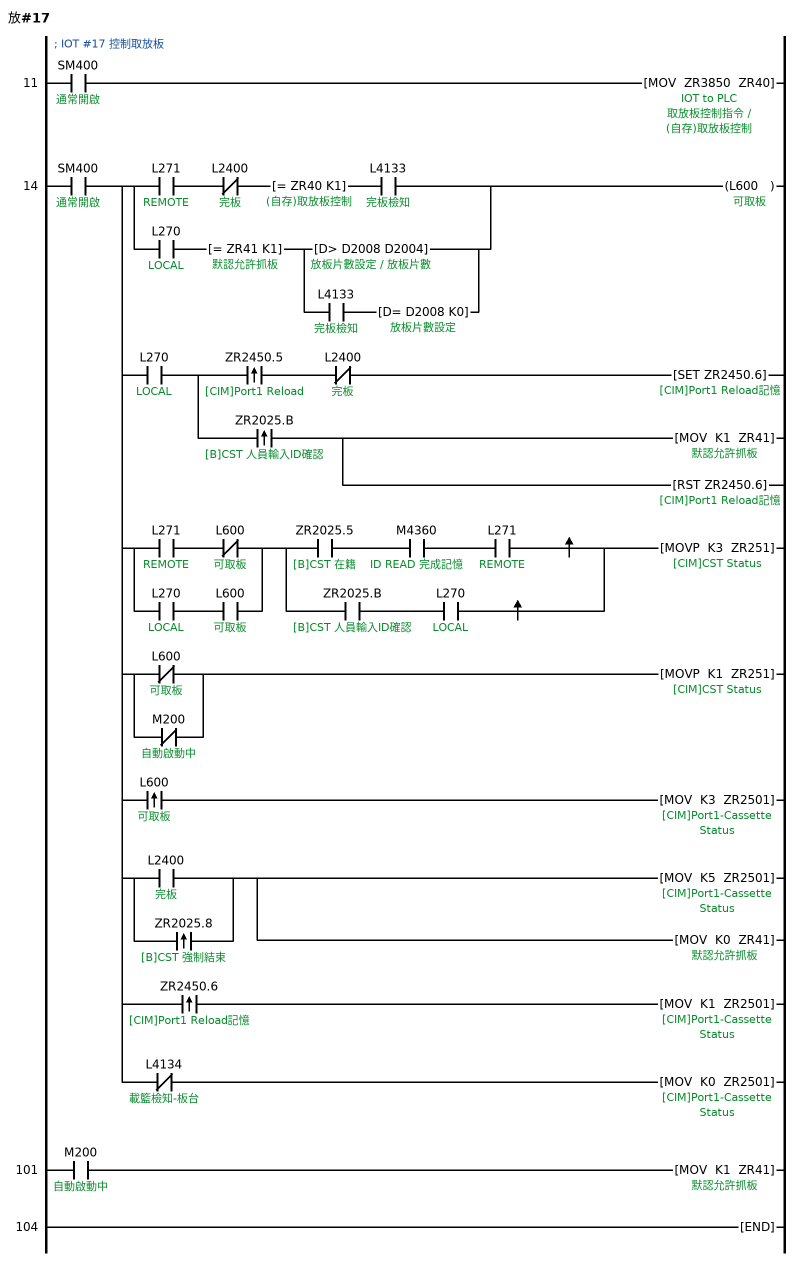
; IOT #17 控制取放板
11    LD      SM400  ; 通常開啟
      MOV     ZR3850 ZR40  ; IOT to PLC 取放板控制指令 / (自存)取放板控制
14    LD      SM400  ; 通常開啟
      MPS
      LD      L271  ; REMOTE
      ANI     L2400  ; 完板
      AND=    ZR40 K1  ; (自存)取放板控制
      AND     L4133  ; 完板檢知
      LD      L270  ; LOCAL
      AND=    ZR41 K1  ; 默認允許抓板
      LDD>    D2008 D2004  ; 放板片數設定 / 放板片數
      LD      L4133  ; 完板檢知
      ANDD=   D2008 K0  ; 放板片數設定
      ORB
      ANB
      ORB
      ANB
      OUT     L600  ; 可取板
      MRD
      AND     L270  ; LOCAL
      MPS
      ANDP    ZR2450.5  ; [CIM]Port1 Reload
      ANI     L2400  ; 完板
      SET     ZR2450.6  ; [CIM]Port1 Reload記憶
      MPP
      ANDP    ZR2025.B  ; [B]CST 人員輸入ID確認
      MOV     K1 ZR41
      RST     ZR2450.6  ; [CIM]Port1 Reload記憶
      MRD
      LD      L271  ; REMOTE
      ANI     L600  ; 可取板
      LD      L270  ; LOCAL
      AND     L600  ; 可取板
      ORB
      ANB
      LD      ZR2025.5  ; [B]CST 在籍
      AND     M4360  ; ID READ 完成記憶
      AND     L271  ; REMOTE
      MEP
      LD      ZR2025.B  ; [B]CST 人員輸入ID確認
      AND     L270  ; LOCAL
      MEP
      ORB
      ANB
      MOVP    K3 ZR251  ; [CIM]CST Status
      MRD
      LDI     L600  ; 可取板
      ORI     M200  ; 自動啟動中
      ANB
      MOVP    K1 ZR251
      MRD
      ANDP    L600  ; 可取板
      MOV     K3 ZR2501  ; [CIM]Port1-Cassette Status
      MRD
      LD      L2400  ; 完板
      ORP     ZR2025.8  ; [B]CST 強制結束
      ANB
      MOV     K5 ZR2501
      MOV     K0 ZR41
      MRD
      ANDP    ZR2450.6  ; [CIM]Port1 Reload記憶
      MOV     K1 ZR2501
      MPP
      ANI     L4134  ; 載籃檢知-板台
      MOV     K0 ZR2501
101   LD      M200  ; 自動啟動中
      MOV     K1 ZR41
104   END
END_PROGRAM

PROGRAM M98
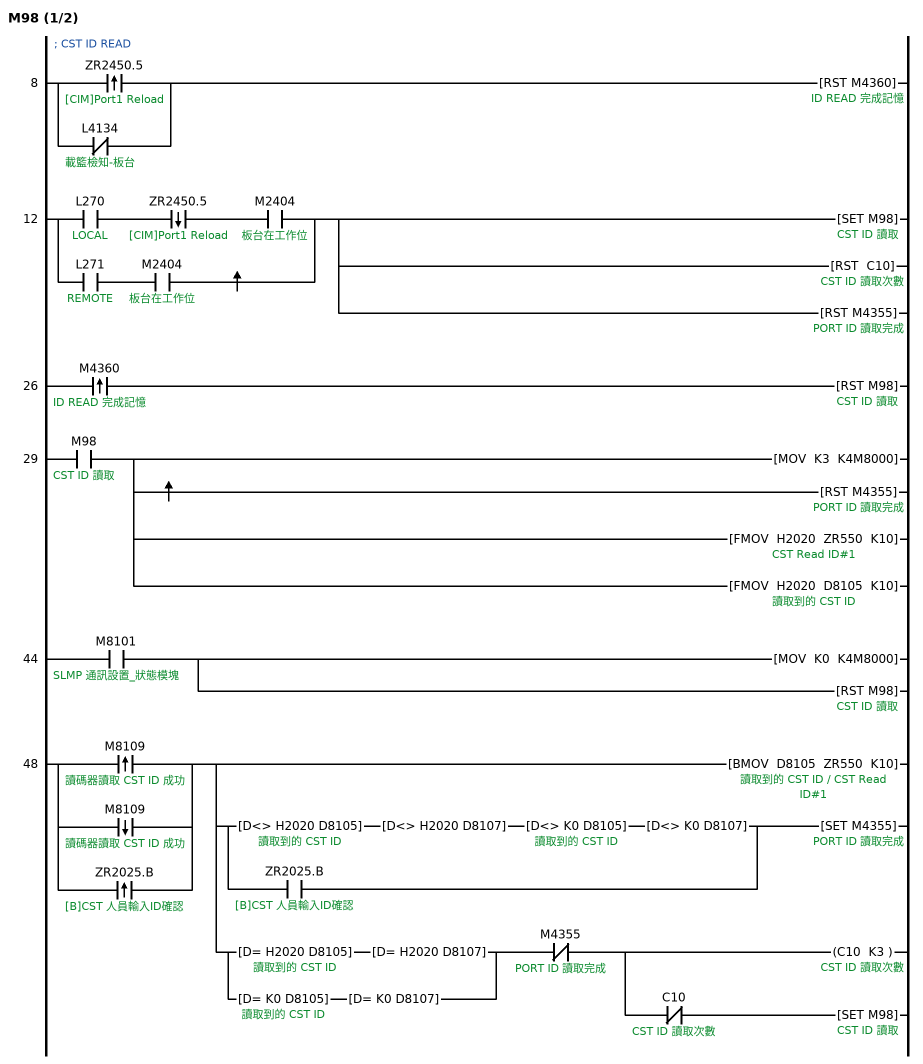
; CST ID READ
8     LDP     ZR2450.5  ; [CIM]Port1 Reload
      ORI     L4134  ; 載籃檢知-板台
      RST     M4360  ; ID READ 完成記憶
12    LD      L270  ; LOCAL
      ANDF    ZR2450.5  ; [CIM]Port1 Reload
      AND     M2404  ; 板台在工作位
      LD      L271  ; REMOTE
      AND     M2404  ; 板台在工作位
      MEP
      ORB
      SET     M98  ; CST ID 讀取
      RST     C10  ; CST ID 讀取次數
      RST     M4355  ; PORT ID 讀取完成
26    LDP     M4360  ; ID READ 完成記憶
      RST     M98  ; CST ID 讀取
29    LD      M98  ; CST ID 讀取
      MOV     K3 K4M8000  ; SLMP 通訊設置_控制模塊
      MPS
      MEP
      RST     M4355  ; PORT ID 讀取完成
      MPP
      FMOV    H2020 ZR550 K10  ; CST Read ID#1
      FMOV    H2020 D8105 K10  ; 讀取到的 CST ID
44    LD      M8101  ; SLMP 通訊設置_狀態模塊
      MOV     K0 K4M8000
      RST     M98  ; CST ID 讀取
48    LDP     M8109  ; 讀碼器讀取 CST ID 成功
      ORF     M8109  ; 讀碼器讀取 CST ID 成功
      ORP     ZR2025.B  ; [B]CST 人員輸入ID確認
      BMOV    D8105 ZR550 K10
      MPS
      LDD<>   H2020 D8105  ; 讀取到的 CST ID
      ANDD<>  H2020 D8107
      ANDD<>  K0 D8105  ; 讀取到的 CST ID
      ANDD<>  K0 D8107
      OR      ZR2025.B  ; [B]CST 人員輸入ID確認
      ANB
      SET     M4355  ; PORT ID 讀取完成
      MPP
      LDD=    H2020 D8105  ; 讀取到的 CST ID
      ANDD=   H2020 D8107
      LDD=    K0 D8105  ; 讀取到的 CST ID
      ANDD=   K0 D8107
      ORB
      ANB
      ANI     M4355  ; PORT ID 讀取完成
      OUT     C10 K3  ; CST ID 讀取次數
      ANI     C10  ; CST ID 讀取次數
      SET     M98  ; CST ID 讀取
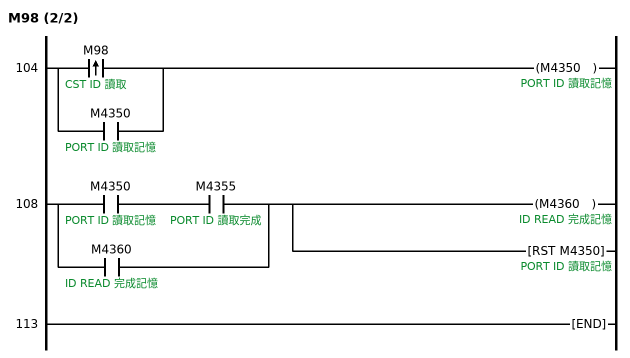
104   LDP     M98  ; CST ID 讀取
      OR      M4350  ; PORT ID 讀取記憶
      OUT     M4350  ; PORT ID 讀取記憶
108   LD      M4350  ; PORT ID 讀取記憶
      AND     M4355  ; PORT ID 讀取完成
      OR      M4360  ; ID READ 完成記憶
      OUT     M4360  ; ID READ 完成記憶
      RST     M4350  ; PORT ID 讀取記憶
113   END
END_PROGRAM

PROGRAM 低M90
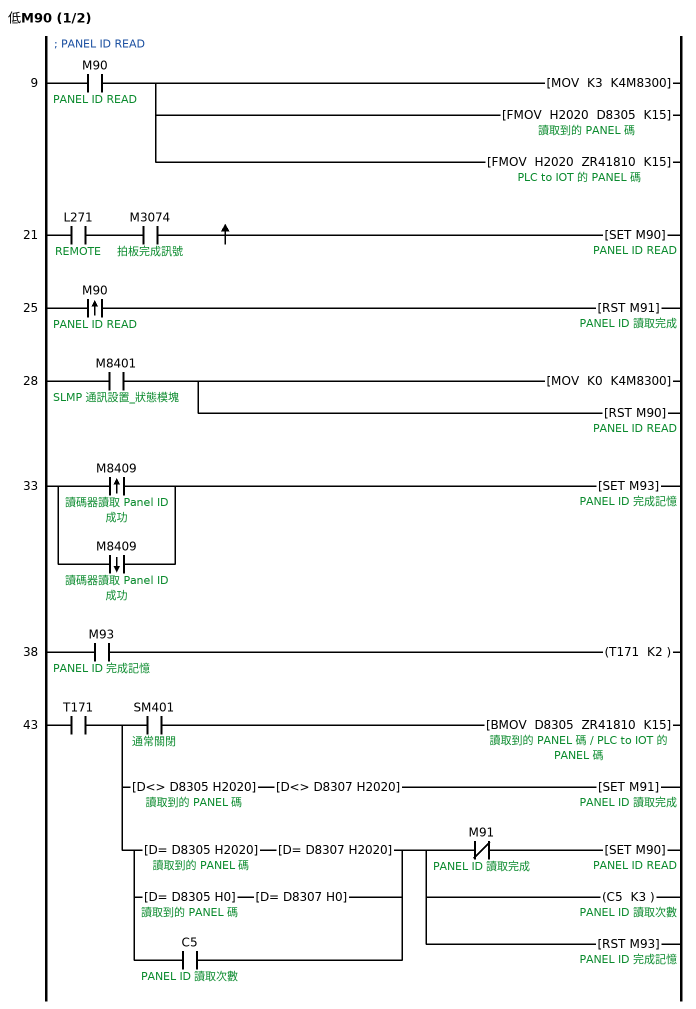
; PANEL ID READ
9     LD      M90  ; PANEL ID READ
      MOV     K3 K4M8300  ; SLMP 通訊設置_控制模塊
      FMOV    H2020 D8305 K15  ; 讀取到的 PANEL 碼
      FMOV    H2020 ZR41810 K15  ; PLC to IOT 的 PANEL 碼
21    LD      L271  ; REMOTE
      AND     M3074  ; 拍板完成訊號
      MEP
      SET     M90  ; PANEL ID READ
25    LDP     M90  ; PANEL ID READ
      RST     M91  ; PANEL ID 讀取完成
28    LD      M8401  ; SLMP 通訊設置_狀態模塊
      MOV     K0 K4M8300
      RST     M90  ; PANEL ID READ
33    LDP     M8409  ; 讀碼器讀取 Panel ID 成功
      ORF     M8409  ; 讀碼器讀取 Panel ID 成功
      SET     M93  ; PANEL ID 完成記憶
38    LD      M93  ; PANEL ID 完成記憶
      OUT     T171 K2
43    LD      T171
      MPS
      AND     SM401  ; 通常關閉
      BMOV    D8305 ZR41810 K15
      MRD
      ANDD<>  D8305 H2020  ; 讀取到的 PANEL 碼
      ANDD<>  D8307 H2020
      SET     M91  ; PANEL ID 讀取完成
      MPP
      LDD=    D8305 H2020  ; 讀取到的 PANEL 碼
      ANDD=   D8307 H2020
      LDD=    D8305 H0  ; 讀取到的 PANEL 碼
      ANDD=   D8307 H0
      ORB
      OR      C5  ; PANEL ID 讀取次數
      ANB
      MPS
      ANI     M91  ; PANEL ID 讀取完成
      SET     M90  ; PANEL ID READ
      MPP
      OUT     C5 K3  ; PANEL ID 讀取次數
      RST     M93  ; PANEL ID 完成記憶
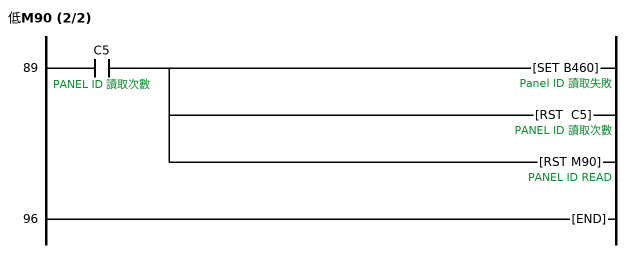
89    LD      C5  ; PANEL ID 讀取次數
      SET     B460  ; Panel ID 讀取失敗
      RST     C5  ; PANEL ID 讀取次數
      RST     M90  ; PANEL ID READ
96    END
END_PROGRAM

PROGRAM 高M90
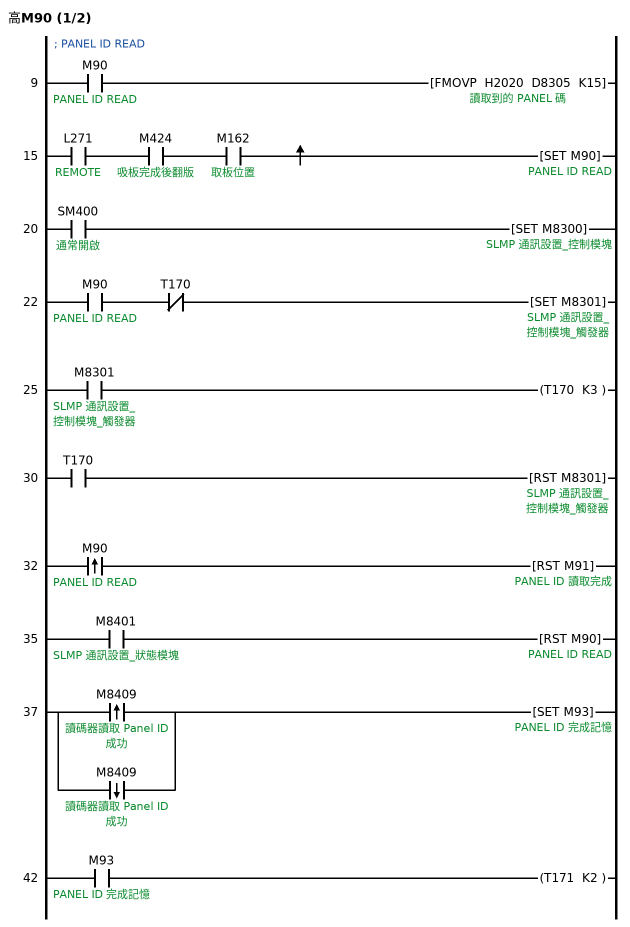
; PANEL ID READ
9     LD      M90  ; PANEL ID READ
      FMOVP   H2020 D8305 K15  ; 讀取到的 PANEL 碼
15    LD      L271  ; REMOTE
      AND     M424  ; 吸板完成後翻版
      AND     M162  ; 取板位置
      MEP
      SET     M90  ; PANEL ID READ
20    LD      SM400  ; 通常開啟
      SET     M8300  ; SLMP 通訊設置_控制模塊
22    LD      M90  ; PANEL ID READ
      ANI     T170
      SET     M8301  ; SLMP 通訊設置_控制模塊_觸發器
25    LD      M8301  ; SLMP 通訊設置_控制模塊_觸發器
      OUT     T170 K3
30    LD      T170
      RST     M8301  ; SLMP 通訊設置_控制模塊_觸發器
32    LDP     M90  ; PANEL ID READ
      RST     M91  ; PANEL ID 讀取完成
35    LD      M8401  ; SLMP 通訊設置_狀態模塊
      RST     M90  ; PANEL ID READ
37    LDP     M8409  ; 讀碼器讀取 Panel ID 成功
      ORF     M8409  ; 讀碼器讀取 Panel ID 成功
      SET     M93  ; PANEL ID 完成記憶
42    LD      M93  ; PANEL ID 完成記憶
      OUT     T171 K2
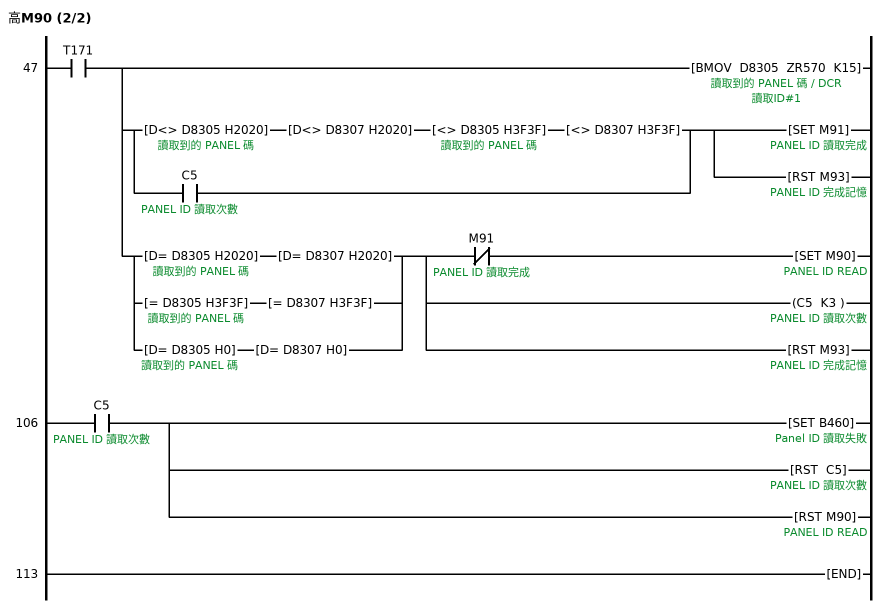
47    LD      T171
      BMOV    D8305 ZR570 K15  ; DCR 讀取ID#1
      MPS
      LDD<>   D8305 H2020  ; 讀取到的 PANEL 碼
      ANDD<>  D8307 H2020
      AND<>   D8305 H3F3F  ; 讀取到的 PANEL 碼
      AND<>   D8307 H3F3F
      OR      C5  ; PANEL ID 讀取次數
      ANB
      SET     M91  ; PANEL ID 讀取完成
      RST     M93  ; PANEL ID 完成記憶
      MPP
      LDD=    D8305 H2020  ; 讀取到的 PANEL 碼
      ANDD=   D8307 H2020
      LD=     D8305 H3F3F  ; 讀取到的 PANEL 碼
      AND=    D8307 H3F3F
      ORB
      LDD=    D8305 H0  ; 讀取到的 PANEL 碼
      ANDD=   D8307 H0
      ORB
      ANB
      MPS
      ANI     M91  ; PANEL ID 讀取完成
      SET     M90  ; PANEL ID READ
      MPP
      OUT     C5 K3  ; PANEL ID 讀取次數
      RST     M93  ; PANEL ID 完成記憶
106   LD      C5  ; PANEL ID 讀取次數
      SET     B460  ; Panel ID 讀取失敗
      RST     C5  ; PANEL ID 讀取次數
      RST     M90  ; PANEL ID READ
113   END
END_PROGRAM

PROGRAM M350
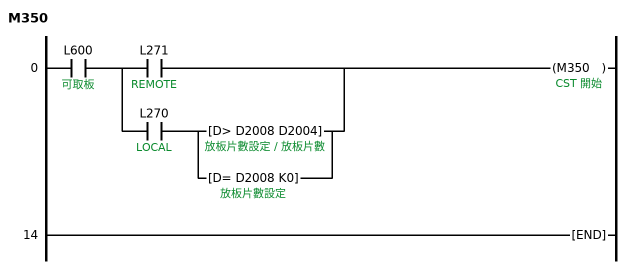
0     LD      L600  ; 可取板
      LD      L271  ; REMOTE
      LD      L270  ; LOCAL
      LDD>    D2008 D2004  ; 放板片數設定 / 放板片數
      ORD=    D2008 K0  ; 放板片數設定
      ANB
      ORB
      ANB
      OUT     M350  ; CST 開始
14    END
END_PROGRAM

PROGRAM M350例
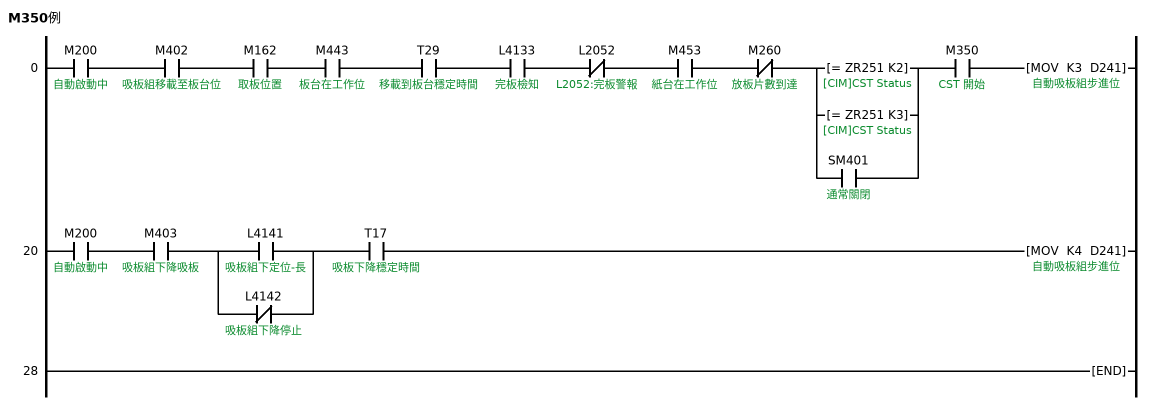
0     LD      M200  ; 自動啟動中
      AND     M402  ; 吸板組移載至板台位
      AND     M162  ; 取板位置
      AND     M443  ; 板台在工作位
      AND     T29  ; 移載到板台穩定時間
      AND     L4133  ; 完板檢知
      ANI     L2052  ; L2052:完板警報
      AND     M453  ; 紙台在工作位
      ANI     M260  ; 放板片數到達
      LD=     ZR251 K2  ; [CIM]CST Status
      OR=     ZR251 K3  ; [CIM]CST Status
      OR      SM401  ; 通常關閉
      ANB
      AND     M350  ; CST 開始
      MOV     K3 D241  ; 自動吸板組步進位
20    LD      M200  ; 自動啟動中
      AND     M403  ; 吸板組下降吸板
      LD      L4141  ; 吸板組下定位-長
      ORI     L4142  ; 吸板組下降停止
      ANB
      AND     T17  ; 吸板下降穩定時間
      MOV     K4 D241
28    END
END_PROGRAM

PROGRAM 中#14
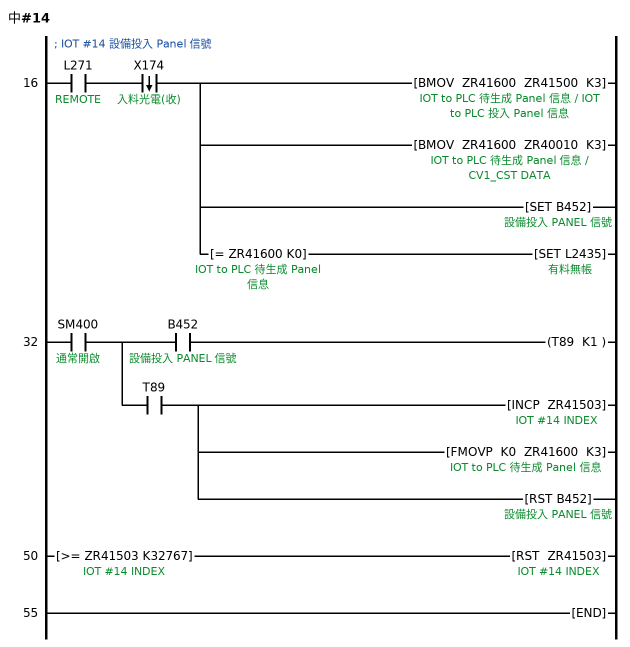
; IOT #14 設備投入 Panel 信號
16    LD      L271  ; REMOTE
      ANDF    X174  ; 入料光電(收)
      BMOV    ZR41600 ZR41500 K3  ; IOT to PLC 待生成 Panel 信息 / IOT to PLC 投入 Panel 信息
      BMOV    ZR41600 ZR40010 K3  ; CV1_CST DATA
      SET     B452  ; 設備投入 PANEL 信號
      AND=    ZR41600 K0  ; IOT to PLC 待生成 Panel 信息
      SET     L2435  ; 有料無帳
32    LD      SM400  ; 通常開啟
      MPS
      AND     B452  ; 設備投入 PANEL 信號
      OUT     T89 K1
      MPP
      AND     T89
      INCP    ZR41503  ; IOT #14 INDEX
      FMOVP   K0 ZR41600 K3
      RST     B452  ; 設備投入 PANEL 信號
50    LD>=    ZR41503 K32767  ; IOT #14 INDEX
      RST     ZR41503  ; IOT #14 INDEX
55    END
END_PROGRAM

PROGRAM 中#15
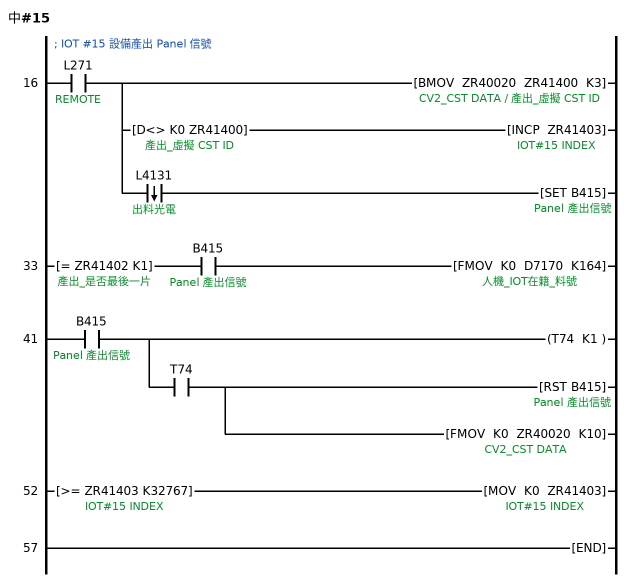
; IOT #15 設備產出 Panel 信號
16    LD      L271  ; REMOTE
      BMOV    ZR40020 ZR41400 K3  ; CV2_CST DATA / 產出_虛擬 CST ID
      MPS
      ANDD<>  K0 ZR41400  ; 產出_虛擬 CST ID
      INCP    ZR41403  ; IOT#15 INDEX
      MPP
      ANDF    L4131  ; 出料光電
      SET     B415  ; Panel 產出信號
33    LD=     ZR41402 K1  ; 產出_是否最後一片
      AND     B415  ; Panel 產出信號
      FMOV    K0 D7170 K164  ; 人機_IOT在籍_料號
41    LD      B415  ; Panel 產出信號
      OUT     T74 K1
      AND     T74
      RST     B415  ; Panel 產出信號
      FMOV    K0 ZR40020 K10
52    LD>=    ZR41403 K32767  ; IOT#15 INDEX
      MOV     K0 ZR41403
57    END
END_PROGRAM

PROGRAM 中#12#13
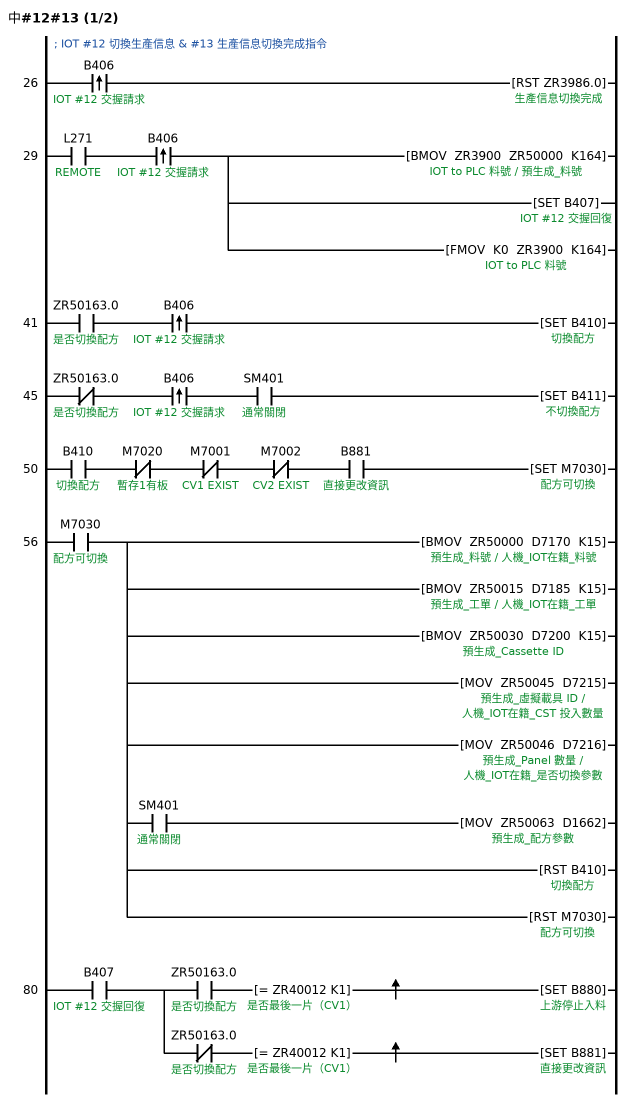
; IOT #12 切換生產信息 & #13 生產信息切換完成指令
26    LDP     B406  ; IOT #12 交握請求
      RST     ZR3986.0  ; 生產信息切換完成
29    LD      L271  ; REMOTE
      ANDP    B406  ; IOT #12 交握請求
      BMOV    ZR3900 ZR50000 K164  ; IOT to PLC 料號 / 預生成_料號
      SET     B407  ; IOT #12 交握回復
      FMOV    K0 ZR3900 K164
41    LD      ZR50163.0  ; 是否切換配方
      ANDP    B406  ; IOT #12 交握請求
      SET     B410  ; 切換配方
45    LDI     ZR50163.0  ; 是否切換配方
      ANDP    B406  ; IOT #12 交握請求
      AND     SM401  ; 通常關閉
      SET     B411  ; 不切換配方
50    LD      B410  ; 切換配方
      ANI     M7020  ; 暫存1有板
      ANI     M7001  ; CV1 EXIST
      ANI     M7002  ; CV2 EXIST
      AND     B881  ; 直接更改資訊
      SET     M7030  ; 配方可切換
56    LD      M7030  ; 配方可切換
      BMOV    ZR50000 D7170 K15  ; 人機_IOT在籍_料號
      BMOV    ZR50015 D7185 K15  ; 預生成_工單 / 人機_IOT在籍_工單
      BMOV    ZR50030 D7200 K15  ; 預生成_Cassette ID
      MOV     ZR50045 D7215  ; 預生成_虛擬載具 ID / 人機_IOT在籍_CST 投入數量
      MOV     ZR50046 D7216  ; 預生成_Panel 數量 / 人機_IOT在籍_是否切換參數
      MPS
      AND     SM401  ; 通常關閉
      MOV     ZR50063 D1662  ; 預生成_配方參數
      MPP
      RST     B410  ; 切換配方
      RST     M7030  ; 配方可切換
80    LD      B407  ; IOT #12 交握回復
      MPS
      AND     ZR50163.0  ; 是否切換配方
      AND=    ZR40012 K1  ; 是否最後一片（CV1）
      MEP
      SET     B880  ; 上游停止入料
      MPP
      ANI     ZR50163.0  ; 是否切換配方
      AND=    ZR40012 K1  ; 是否最後一片（CV1）
      MEP
      SET     B881  ; 直接更改資訊
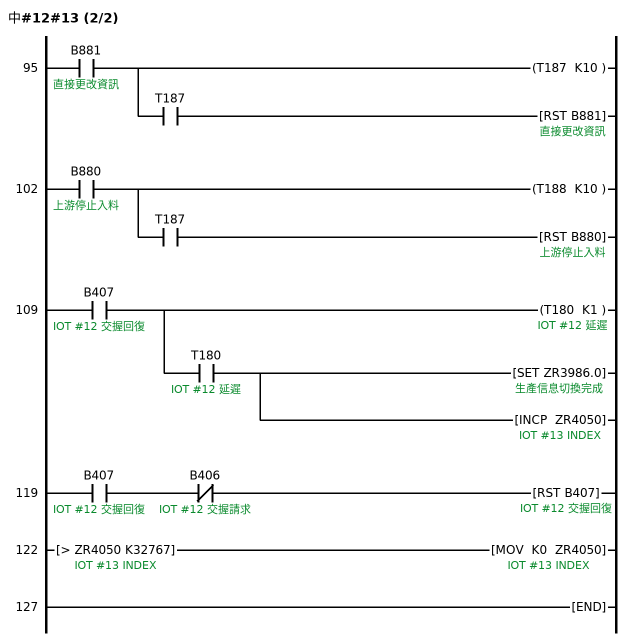
95    LD      B881  ; 直接更改資訊
      OUT     T187 K10
      AND     T187
      RST     B881  ; 直接更改資訊
102   LD      B880  ; 上游停止入料
      OUT     T188 K10
      AND     T187
      RST     B880  ; 上游停止入料
109   LD      B407  ; IOT #12 交握回復
      OUT     T180 K1  ; IOT #12 延遲
      AND     T180  ; IOT #12 延遲
      SET     ZR3986.0  ; 生產信息切換完成
      INCP    ZR4050  ; IOT #13 INDEX
119   LD      B407  ; IOT #12 交握回復
      ANI     B406  ; IOT #12 交握請求
      RST     B407  ; IOT #12 交握回復
122   LD>     ZR4050 K32767  ; IOT #13 INDEX
      MOV     K0 ZR4050
127   END
END_PROGRAM

PROGRAM 附
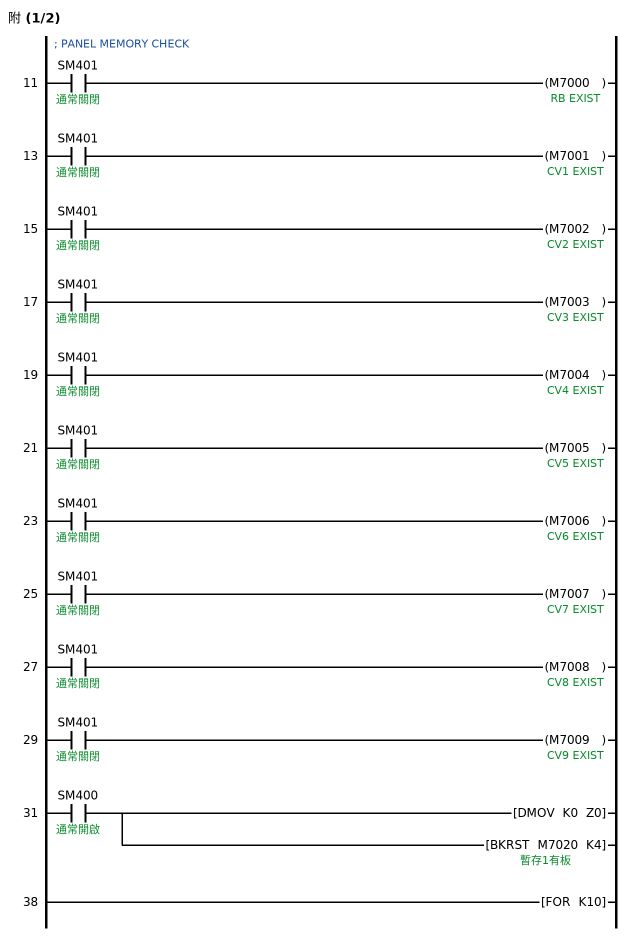
; PANEL MEMORY CHECK
11    LD      SM401  ; 通常關閉
      OUT     M7000  ; RB EXIST
13    LD      SM401  ; 通常關閉
      OUT     M7001  ; CV1 EXIST
15    LD      SM401  ; 通常關閉
      OUT     M7002  ; CV2 EXIST
17    LD      SM401  ; 通常關閉
      OUT     M7003  ; CV3 EXIST
19    LD      SM401  ; 通常關閉
      OUT     M7004  ; CV4 EXIST
21    LD      SM401  ; 通常關閉
      OUT     M7005  ; CV5 EXIST
23    LD      SM401  ; 通常關閉
      OUT     M7006  ; CV6 EXIST
25    LD      SM401  ; 通常關閉
      OUT     M7007  ; CV7 EXIST
27    LD      SM401  ; 通常關閉
      OUT     M7008  ; CV8 EXIST
29    LD      SM401  ; 通常關閉
      OUT     M7009  ; CV9 EXIST
31    LD      SM400  ; 通常開啟
      DMOV    K0 Z0
      BKRST   M7020 K4  ; 暫存1有板
38    FOR     K10
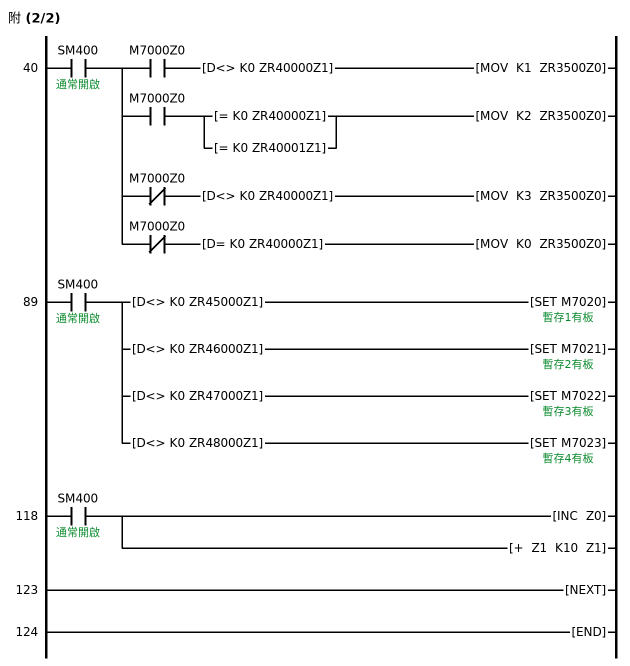
40    LD      SM400  ; 通常開啟
      MPS
      AND     M7000Z0
      ANDD<>  K0 ZR40000Z1
      MOV     K1 ZR3500Z0
      MRD
      AND     M7000Z0
      LD=     K0 ZR40000Z1
      OR=     K0 ZR40001Z1
      ANB
      MOV     K2 ZR3500Z0
      MRD
      ANI     M7000Z0
      ANDD<>  K0 ZR40000Z1
      MOV     K3 ZR3500Z0
      MPP
      ANI     M7000Z0
      ANDD=   K0 ZR40000Z1
      MOV     K0 ZR3500Z0
89    LD      SM400  ; 通常開啟
      MPS
      ANDD<>  K0 ZR45000Z1
      SET     M7020  ; 暫存1有板
      MRD
      ANDD<>  K0 ZR46000Z1
      SET     M7021  ; 暫存2有板
      MRD
      ANDD<>  K0 ZR47000Z1
      SET     M7022  ; 暫存3有板
      MPP
      ANDD<>  K0 ZR48000Z1
      SET     M7023  ; 暫存4有板
118   LD      SM400  ; 通常開啟
      INC     Z0
      +       Z1 K10 Z1
123   NEXT
124   END
END_PROGRAM

PROGRAM FIFO
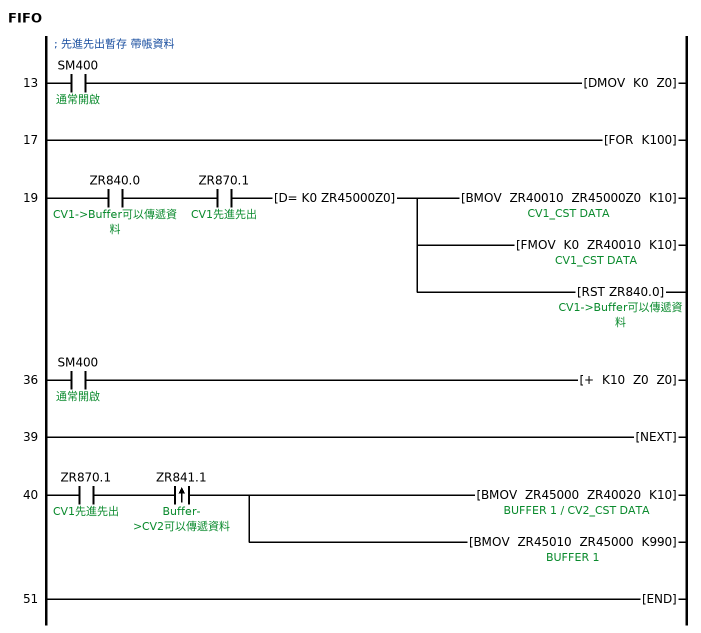
; 先進先出暫存 帶帳資料
13    LD      SM400  ; 通常開啟
      DMOV    K0 Z0
17    FOR     K100
19    LD      ZR840.0  ; CV1->Buffer可以傳遞資料
      AND     ZR870.1  ; CV1先進先出
      ANDD=   K0 ZR45000Z0
      BMOV    ZR40010 ZR45000Z0 K10  ; CV1_CST DATA
      FMOV    K0 ZR40010 K10
      RST     ZR840.0  ; CV1->Buffer可以傳遞資料
36    LD      SM400  ; 通常開啟
      +       K10 Z0 Z0
39    NEXT
40    LD      ZR870.1  ; CV1先進先出
      ANDP    ZR841.1  ; Buffer->CV2可以傳遞資料
      BMOV    ZR45000 ZR40020 K10  ; BUFFER 1 / CV2_CST DATA
      BMOV    ZR45010 ZR45000 K990
51    END
END_PROGRAM

PROGRAM FILO
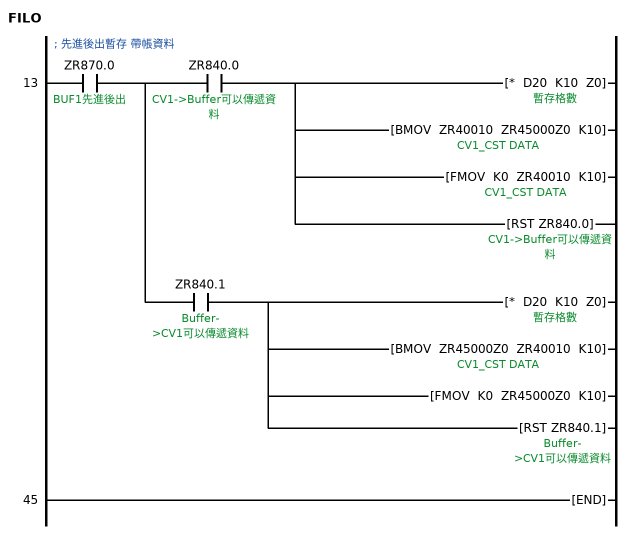
; 先進後出暫存 帶帳資料
13    LD      ZR870.0  ; BUF1先進後出
      MPS
      AND     ZR840.0  ; CV1->Buffer可以傳遞資料
      *       D20 K10 Z0  ; 暫存格數
      BMOV    ZR40010 ZR45000Z0 K10  ; CV1_CST DATA
      FMOV    K0 ZR40010 K10
      RST     ZR840.0  ; CV1->Buffer可以傳遞資料
      MPP
      AND     ZR840.1  ; Buffer->CV1可以傳遞資料
      *       D20 K10 Z0
      BMOV    ZR45000Z0 ZR40010 K10
      FMOV    K0 ZR45000Z0 K10
      RST     ZR840.1  ; Buffer->CV1可以傳遞資料
45    END
END_PROGRAM

PROGRAM FILO#16
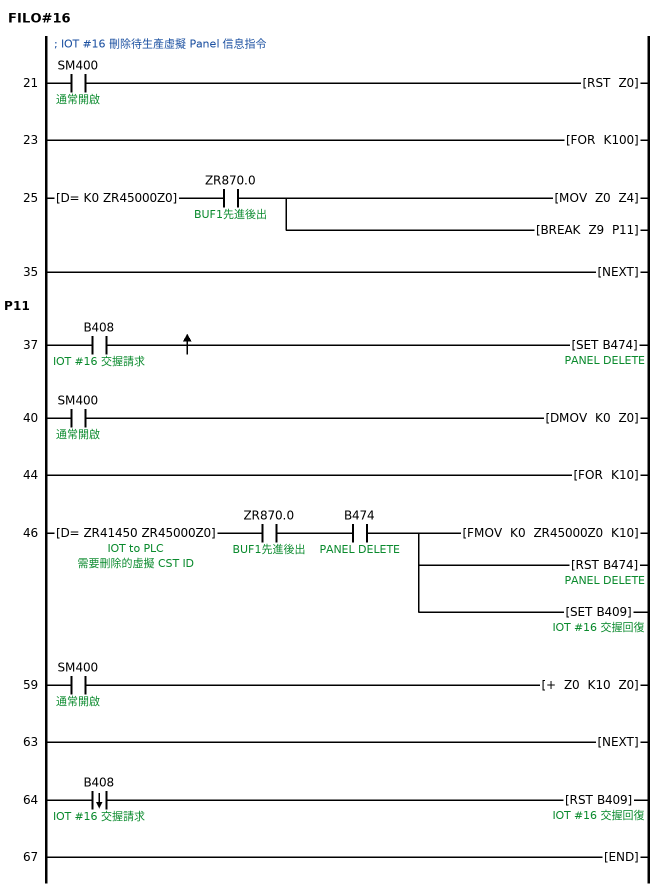
; IOT #16 刪除待生產虛擬 Panel 信息指令
21    LD      SM400  ; 通常開啟
      RST     Z0
23    FOR     K100
25    LDD=    K0 ZR45000Z0
      AND     ZR870.0  ; BUF1先進後出
      MOV     Z0 Z4
      BREAK   Z9 P11
35    NEXT
      P11
37    LD      B408  ; IOT #16 交握請求
      MEP
      SET     B474  ; PANEL DELETE
40    LD      SM400  ; 通常開啟
      DMOV    K0 Z0
44    FOR     K10
46    LDD=    ZR41450 ZR45000Z0  ; IOT to PLC 需要刪除的虛擬 CST ID
      AND     ZR870.0  ; BUF1先進後出
      AND     B474  ; PANEL DELETE
      FMOV    K0 ZR45000Z0 K10
      RST     B474  ; PANEL DELETE
      SET     B409  ; IOT #16 交握回復
59    LD      SM400  ; 通常開啟
      +       Z0 K10 Z0
63    NEXT
64    LDF     B408  ; IOT #16 交握請求
      RST     B409  ; IOT #16 交握回復
67    END
END_PROGRAM

PROGRAM FIFO#16
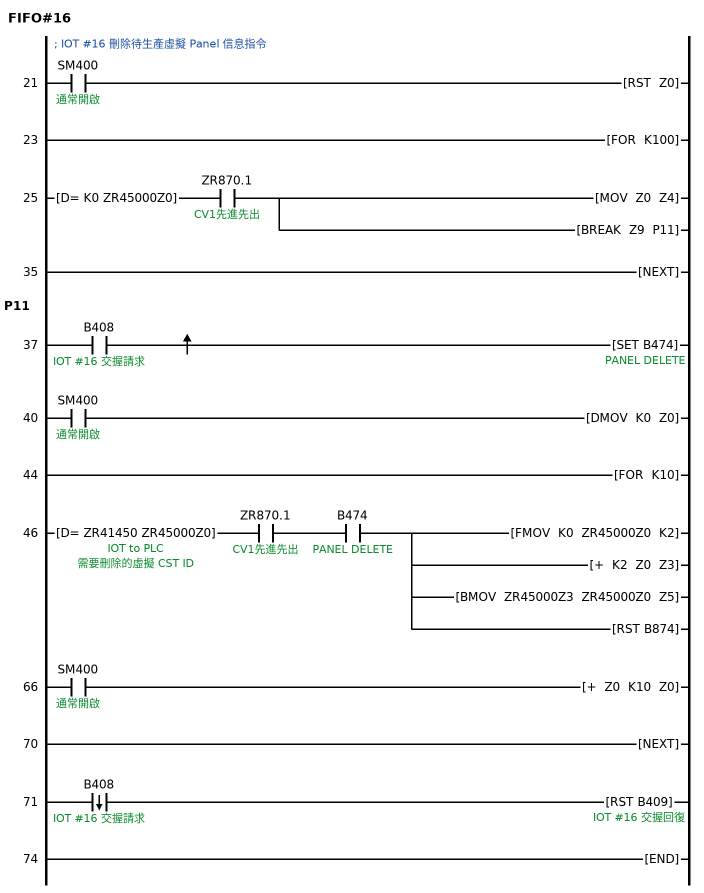
; IOT #16 刪除待生產虛擬 Panel 信息指令
21    LD      SM400  ; 通常開啟
      RST     Z0
23    FOR     K100
25    LDD=    K0 ZR45000Z0
      AND     ZR870.1  ; CV1先進先出
      MOV     Z0 Z4
      BREAK   Z9 P11
35    NEXT
      P11
37    LD      B408  ; IOT #16 交握請求
      MEP
      SET     B474  ; PANEL DELETE
40    LD      SM400  ; 通常開啟
      DMOV    K0 Z0
44    FOR     K10
46    LDD=    ZR41450 ZR45000Z0  ; IOT to PLC 需要刪除的虛擬 CST ID
      AND     ZR870.1  ; CV1先進先出
      AND     B474  ; PANEL DELETE
      FMOV    K0 ZR45000Z0 K2
      +       K2 Z0 Z3
      BMOV    ZR45000Z3 ZR45000Z0 Z5
      RST     B874
66    LD      SM400  ; 通常開啟
      +       Z0 K10 Z0
70    NEXT
71    LDF     B408  ; IOT #16 交握請求
      RST     B409  ; IOT #16 交握回復
74    END
END_PROGRAM

// device comments not shown above
ZR40011  ; CV1_PANEL DATA
ZR40021  ; CV2_PANEL DATA
ZR40022  ; 是否最後一片（CV2）
ZR40030  ; CV3_CST DATA
ZR40031  ; CV3_PANEL DATA
ZR40032  ; 是否最後一片（CV3）
ZR40040  ; CV4_CST DATA
ZR40041  ; CV4_PANEL DATA
ZR40042  ; 是否最後一片（CV4）
ZR40050  ; CV5_CST DATA
ZR40051  ; CV5_PANEL DATA
ZR40052  ; 是否最後一片（CV5）
ZR40060  ; CV6_CST DATA
ZR40061  ; CV6_PANEL DATA
ZR40062  ; 是否最後一片（CV6）
ZR40070  ; CV7_CST DATA
ZR40071  ; CV7_PANEL DATA
ZR40072  ; 是否最後一片（CV7）
ZR40080  ; CV8_CST DATA
ZR40081  ; CV8_PANEL DATA
ZR40082  ; 是否最後一片（CV8）
ZR40090  ; CV9_CST DATA
ZR40091  ; CV9_PANEL DATA
ZR40092  ; 是否最後一片（CV9）
ZR45001  ; BUFFER2
ZR45002  ; BUFFER3
ZR45003  ; BUFFER4
ZR46000  ; BUFFER 2
ZR47000  ; BUFFER 3
ZR48000  ; BUFFER 4
